// TIA Portal V19 export
ORGANIZATION_BLOCK "Main"   // OB1, LAD, ProgramCycle
TITLE = "Main Program Sweep (Cycle)"
{ S7_Optimized_Access := 'TRUE' }
// stored: SetENOAutomatically false
   VAR_INPUT
      Initial_Call : Bool;   // Initial call of this OB
      Remanence : Bool;   // =True, if remanent data are available
   END_VAR
   VAR_TEMP   // added for the SCL form of the ladder/FBD networks
      _w1 : Bool;
      _w2 : Bool;
      _w3 : Bool;
      _w4 : Bool;
      _w5 : Bool;
      _w6 : Bool;
      _w7 : Bool;
      _w8 : Bool;
      _w9 : Bool;
      _w10 : Bool;
      _w11 : Bool;
      _w12 : Bool;
      _w13 : Bool;
      _w14 : Bool;
      _w15 : Bool;
      _w16 : Bool;
      _w17 : Bool;
      _w18 : Bool;
      _w19 : Bool;
      _w20 : Bool;
   END_VAR
BEGIN

REGION Network 1
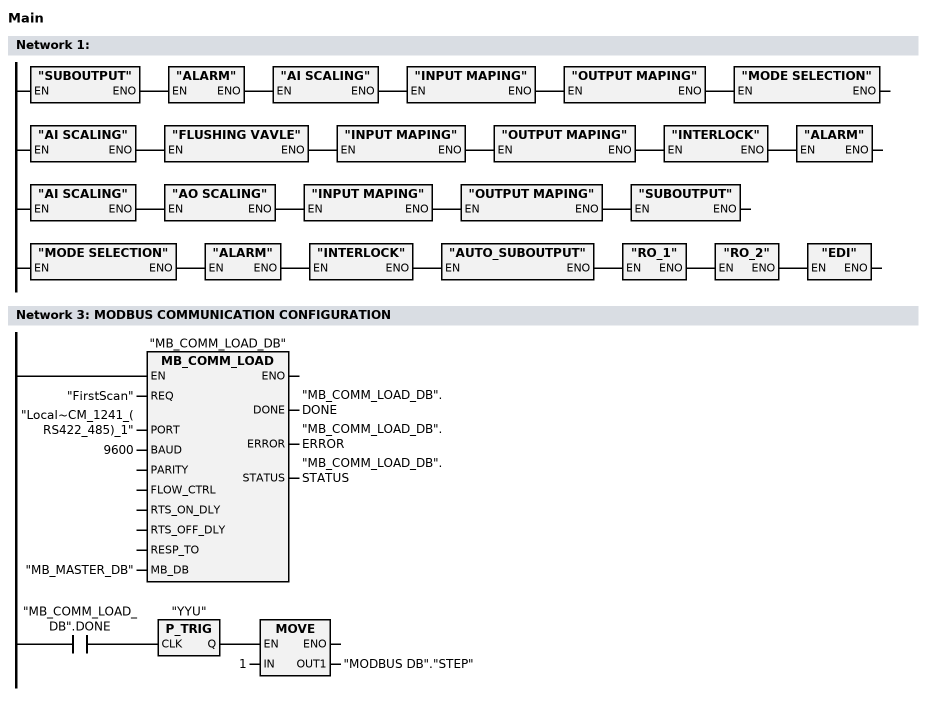
   RUNG wire#powerrail
      "SUBOUTPUT"()
      "ALARM"()
      "AI SCALING"()
      "INPUT MAPING"()
      "OUTPUT MAPING"()
      "MODE SELECTION"()
   END_RUNG
   RUNG wire#powerrail
      "AI SCALING"()
      "FLUSHING VAVLE"()
      "INPUT MAPING"()
      "OUTPUT MAPING"()
      "INTERLOCK"()
      "ALARM"()
   END_RUNG
   RUNG wire#powerrail
      "AI SCALING"()
      "AO SCALING"()
      "INPUT MAPING"()
      "OUTPUT MAPING"()
      "SUBOUTPUT"()
   END_RUNG
   RUNG wire#powerrail
      "MODE SELECTION"()
      "ALARM"()
      "INTERLOCK"()
      "AUTO_SUBOUTPUT"()
      "RO_1"()
      "RO_2"()
      "EDI"()
   END_RUNG
   // the same network as SCL:
   "SUBOUTPUT"(ENO => #_w1);
   "ALARM"(EN := #_w1, ENO => #_w2);
   "AI SCALING"(EN := #_w2, ENO => #_w3);
   "INPUT MAPING"(EN := #_w3, ENO => #_w4);
   "OUTPUT MAPING"(EN := #_w4, ENO => #_w5);
   IF #_w5 THEN "MODE SELECTION"(); END_IF;
   "AI SCALING"(ENO => #_w6);
   "FLUSHING VAVLE"(EN := #_w6, ENO => #_w7);
   "INPUT MAPING"(EN := #_w7, ENO => #_w8);
   "OUTPUT MAPING"(EN := #_w8, ENO => #_w9);
   "INTERLOCK"(EN := #_w9, ENO => #_w10);
   IF #_w10 THEN "ALARM"(); END_IF;
   "AI SCALING"(ENO => #_w11);
   "AO SCALING"(EN := #_w11, ENO => #_w12);
   "INPUT MAPING"(EN := #_w12, ENO => #_w13);
   "OUTPUT MAPING"(EN := #_w13, ENO => #_w14);
   IF #_w14 THEN "SUBOUTPUT"(); END_IF;
   "MODE SELECTION"(ENO => #_w15);
   "ALARM"(EN := #_w15, ENO => #_w16);
   "INTERLOCK"(EN := #_w16, ENO => #_w17);
   "AUTO_SUBOUTPUT"(EN := #_w17, ENO => #_w18);
   "RO_1"(EN := #_w18, ENO => #_w19);
   "RO_2"(EN := #_w19, ENO => #_w20);
   IF #_w20 THEN "EDI"(); END_IF;
END_REGION

REGION Network 3: MODBUS COMMUNICATION CONFIGURATION
   RUNG wire#powerrail
      "MB_COMM_LOAD_DB".MB_COMM_LOAD(REQ := "FirstScan", PORT := "Local~CM_1241_(RS422_485)_1", BAUD := 9600, PARITY :=, FLOW_CTRL :=, RTS_ON_DLY :=, RTS_OFF_DLY :=, RESP_TO :=, MB_DB := "MB_MASTER_DB", DONE => "MB_COMM_LOAD_DB".DONE, ERROR => "MB_COMM_LOAD_DB".ERROR, STATUS => "MB_COMM_LOAD_DB".STATUS)
   END_RUNG
   RUNG wire#powerrail
      Contact( "MB_COMM_LOAD_DB".DONE )
      P_Trig( "YYU" )
      Move(in := 1, out1 => "MODBUS DB"."STEP")
   END_RUNG
   // the same network as SCL:
   "MB_COMM_LOAD_DB"(REQ := "FirstScan",   // MB_COMM_LOAD
                     PORT := "Local~CM_1241_(RS422_485)_1",
                     BAUD := 9600,
                     MB_DB := "MB_MASTER_DB",
                     DONE => "MB_COMM_LOAD_DB".DONE,
                     ERROR => "MB_COMM_LOAD_DB".ERROR,
                     STATUS => "MB_COMM_LOAD_DB".STATUS);
   #_w1 := "MB_COMM_LOAD_DB".DONE AND NOT "YYU";   // rising edge
   "YYU" := "MB_COMM_LOAD_DB".DONE;
   IF #_w1 THEN "MODBUS DB"."STEP" := 1; END_IF;
END_REGION

REGION Network 4: slave plc
END_REGION
END_ORGANIZATION_BLOCK
